TYPE ST_SavedStructure :
STRUCT
	CurrentPos		:	REAL;
	FwdSoftLim		:	REAL;
	RevSoftLim		:	REAL;
	Counter			:	INT;
	SavedPos		:	ARRAY [1..25] OF ST_SavedPositions;
END_STRUCT
END_TYPE

(* stored: Version 1.1.0.1, ProductVersion 3.1.4022.12
   DUT ST_SavedStructure: Id {b7ffbcaa-7c3b-4f1f-ade3-c48f89174665} *)
